{attribute 'linkalways'} 
{attribute 'no_explicit_call' := 'This FB is a CLASS and must be accessed using methods or properties'}
{attribute 'enable_dynamic_creation'}
FUNCTION_BLOCK _ETcVnSvm EXTENDS EnumDatatypeBase
VAR
	localData : ETcVnSvm;
	activeData : REFERENCE TO ETcVnSvm;
	enumBaseDatatype : _UDINT(localData);
END_VAR

METHOD PRIVATE AddLocalEnumeration
VAR_INPUT
	Enumeration : T_MAXSTRING;
	Value : ETcVnSvm;
END_VAR
AddEnumeration(Enumeration, Value);
END_METHOD

PROPERTY PUBLIC Address : PVOID
GET
Address := ADR(activeData);
END_GET
END_PROPERTY

METHOD PUBLIC ClearReference
VAR_INPUT
END_VAR
activeData REF= localData;
SetBaseDatatypeReference();
END_METHOD

METHOD PUBLIC Clone : I_Datatype
VAR
    pClone : POINTER TO _ETcVnSvm;
END_VAR
pClone := __NEW(_ETcVnSvm(InitialValue := Value));
Clone := pClone^;
END_METHOD

METHOD FB_init : BOOL
VAR_INPUT
	bInitRetains : BOOL; // if TRUE, the retain variables are initialized (warm start / cold start)
	bInCopyCode : BOOL;  // if TRUE, the instance afterwards gets moved into the copy code (online change)
	InitialValue : ETcVnSvm;
END_VAR
localData := InitialValue;
AddBaseDatatype(enumBaseDatatype);
ClearReference();

AddLocalEnumeration('TCVN_SVM_C_CLASSIFIER', ETcVnSvm.TCVN_SVM_C_CLASSIFIER);
AddLocalEnumeration('TCVN_SVM_NU_CLASSIFIER', ETcVnSvm.TCVN_SVM_NU_CLASSIFIER);
AddLocalEnumeration('TCVN_SVM_NOVELTY_DETECTOR', ETcVnSvm.TCVN_SVM_NOVELTY_DETECTOR);
AddLocalEnumeration('TCVN_SVM_EPS_REGRESSOR', ETcVnSvm.TCVN_SVM_EPS_REGRESSOR);
AddLocalEnumeration('TCVN_SVM_NU_REGRESSOR', ETcVnSvm.TCVN_SVM_NU_REGRESSOR);
END_METHOD

PROPERTY PUBLIC Identifier : T_MAXSTRING
GET
Identifier := 'ETcVnSvm';
END_GET
END_PROPERTY

METHOD IsEnumeratorValueEqual : BOOL
VAR_INPUT
	Enumerator : I_KeyValueForwardEnumerator;
END_VAR
VAR
	storedValue : ETcVnSvm;
END_VAR
IF NOT Enumerator.TryGet(storedValue) THEN
	RETURN;
END_IF

IsEnumeratorValueEqual := storedValue = activeData;
END_METHOD

METHOD PUBLIC MakeReferenceTo
VAR_INPUT
	ReferenceTarget : REFERENCE TO ETcVnSvm;
END_VAR
activeData REF= ReferenceTarget;
SetBaseDatatypeReference();
END_METHOD

METHOD PROTECTED SetBaseDatatypeReference
VAR_INPUT
END_VAR
enumBaseDatatype.MakeReferenceTo(activeData);
END_METHOD

PROPERTY PUBLIC Size : UDINT
GET
Size := SIZEOF(activeData);
END_GET
END_PROPERTY

METHOD TryMakeReferenceTo : BOOL
VAR_INPUT
	Target : I_Datatype;
END_VAR
VAR
	targetAsEnum : I_EnumDatatype;
	pTargetData : POINTER TO ETcVnSvm;
END_VAR
IF NOT Target.TryResolveAsEnumDatatype(targetAsEnum) THEN
	RETURN;
END_IF

IF targetAsEnum.Identifier <> Identifier THEN
	RETURN;
END_IF

pTargetData := Target.Address;
activeData REF= pTargetData^;
SetBaseDatatypeReference();
TryMakeReferenceTo := TRUE;
END_METHOD

PROPERTY PUBLIC Value : ETcVnSvm
GET
Value := activeData;
END_GET
SET
activeData := Value;
END_SET
END_PROPERTY

END_FUNCTION_BLOCK

(* stored: Version 1.1.0.1, ProductVersion 3.1.4024.12
   POU _ETcVnSvm: Id {9a114354-2072-4cad-9222-bc6e2a685b2d}, SpecialFunc None
   Folder Constructor: Id {f6487f8c-2507-42ea-b5cf-8a517becbd0c}
   Folder Private: Id {6b6e69b2-a494-4b14-b50f-66a3944e2680}
   Folder Protected: Id {092686df-276e-4b9a-9da5-f8286b36326d}
   Method AddLocalEnumeration: Id {166269f7-8de4-40a1-b806-f43e7ce0a998}
   Property Address: Id {477eb0ce-9cec-4711-8772-0c342b8e083e}
   Get Get: Id {a2685c6c-10a4-48cc-ae4e-05c8d860f426}
   Method ClearReference: Id {f43c2937-ae1c-4249-87b3-b9eeefa3a664}
   Method Clone: Id {0ac56021-78cd-4254-bbed-e55513aadf35}
   Method FB_init: Id {561034d0-bdd2-4771-b945-77ab095cfe69}
   Property Identifier: Id {a2aea430-05f9-4548-962f-4ee3ce1f5dbd}
   Get Get: Id {afb9cb0c-11f3-4e78-85a3-e0be7abbb3af}
   Method IsEnumeratorValueEqual: Id {a25ea705-021a-4de2-8c08-2d58ee5086f7}
   Method MakeReferenceTo: Id {93fdf46e-1363-466f-aea9-52790228a48e}
   Method SetBaseDatatypeReference: Id {db6d1569-d34e-4a6a-80d3-b23aeff43371}
   Property Size: Id {a4f328cc-a286-45fc-87f8-65838e04319e}
   Get Get: Id {92be0de9-1e57-4145-b086-1d358e4f8b44}
   Method TryMakeReferenceTo: Id {41e5a207-cdbd-4dd1-93f5-8e8be3712201}
   Property Value: Id {45aa4a5b-5f74-4ef6-853c-2d2fbe83637d}
   Get Get: Id {c246928d-0e9f-4faf-ae39-7d98ce0573f8}
   Set Set: Id {7b9c1493-a450-4b87-ab41-3aea405124ab} *)
